{attribute 'pack_mode' := '2'}
TYPE ST_LIST_NODE_DATA :
STRUCT
  ProcessData     : ST_PROCESS_DATA;  // target data
END_STRUCT
END_TYPE

(* stored: Version 1.1.0.1, ProductVersion 3.1.4026.18
   DUT ST_LIST_NODE_DATA: Id {7b55440d-24d3-455c-bb62-c24c3ebe9c22} *)
